// TIA Portal V17 export
// export: Created 2024-10-17T14:16:18.3999577Z, ExportSetting WithDefaults, DisplayName Totally Integrated Automation Portal, DisplayVersion V17 Update 4, DisplayName TIA Portal Openness, DisplayVersion V17 Update 4, DisplayName TIA Portal Version Control Interface, DisplayVersion V17, DisplayName SINAMICS Startdrive Advanced, DisplayVersion V17 Update2, DisplayName SINAMICS Startdrive G130, G150, S120, S150, SINAMICS MV, S210, DisplayVersion V17 Update2, DisplayName SINAMICS Startdrive G110M, G120, G120C, G120D, G120P, G115D, DisplayVersion V17 Update2, DisplayName STEP 7 Professional, DisplayVersion V17 Update 4, DisplayName STEP 7 Safety, DisplayVersion V17, DisplayName WinCC Advanced / Unified PC, DisplayVersion V17 Update 4
TYPE "LPMLV2022_typeProductData"
TITLE = LPMLV2022_typeProductData
// Support: tech.team.motioncontrol@siemens.com
// stored: IsFailsafeCompliant false
   STRUCT
      ID { ExternalWritable := 'False'} : DInt;   // ID Number for each Product Stream. The product IDs are used to report product identity for each product stream
      "Name" { ExternalWritable := 'False'} : String[80];   // Name of Product Stream. The Name element is used to further report the identity of the product within the product stream, especially when alphanumeric characters are used (i.e. SKU or UPC)
      Unit { ExternalWritable := 'False'} : String[6];   // Unit of Measure of each Product Stream. The Unit element is used to report the unit of production for the product within the product stream. An example product unit of measure may be Pc, Crtn, Case, etc
      PrimaryQty { ExternalWritable := 'False'} : Real;   // Product Primary Quantity Value of each Product Stream. The PrimaryQty element is used to provide a common reference for manufacturing throughput across all the machines on a production line. This element relates the number of Primary Products per Unit for a particular product stream. It can be used as a conversion factor for a local machine reference speed since Command.MachSpeed is given in units of PrimaryProducts/Min
      ConsumedCount { ExternalWritable := 'False'} : DInt;   // Consumed Count of each Product Stream. This tag represents the material used/consumed in the production machine for a particular input or output product stream. An example of tag usage would be the number of bags consumed in a filler, or bagger packaging machine, or the amount of linear length used, or the number caps used
      ProcessedCount { ExternalWritable := 'False'} : DInt;   // Processed Count of each Product Stream. This tag represents the number of products from a particular input or output product stream processed by the production machine. An example of tag usage would be the number of products that were made, including all good and defective products. The number of products processed minus the number of defective products is the number of products actually made by the machine. Minimum required for information/machine monitoring
      DefectiveCount { ExternalWritable := 'False'} : DInt;   // Defective Count of each Product Stream. This tag represents the number of products from a particular input or output product stream that is marked as defective in the production machine, to be used if applicable. An example of tag usage would be the number of products rejected or products that are termed defective. Minimum required for information/machine monitoring
      AccConsumedCount { ExternalWritable := 'False'} : DInt;   // Accumulated Consumption Count of each Product Stream Consumption Since Last Reset. This tag represents the total accumulated material used/consumed in the production machine for a particular input or output product stream
      AccProcessedCount { ExternalWritable := 'False'} : DInt;   // Accumulated Processed Count of each Product Stream Since Last Reset. This tag represents the total accumulated number of products from a particular input or output product stream processed by the production machine. An example of tag usage would be the number of products that were made, including all good and defective products. The number of products processed minus the number of defective products is the number of products actually made by the machine
      AccDefectiveCount { ExternalWritable := 'False'} : DInt;   // Accumulated Defective Count of each Product Stream Since Last Reset. This tag represents the total accumulated number of products from a particular input or output product stream that is marked as defective in the production machine, to be used if applicable. An example of tag usage would be the number of products rejected or products that are termed defective
   END_STRUCT;
END_TYPE
